RoboDK station: Silva_Honores_ProyectoFinal (1).rdk

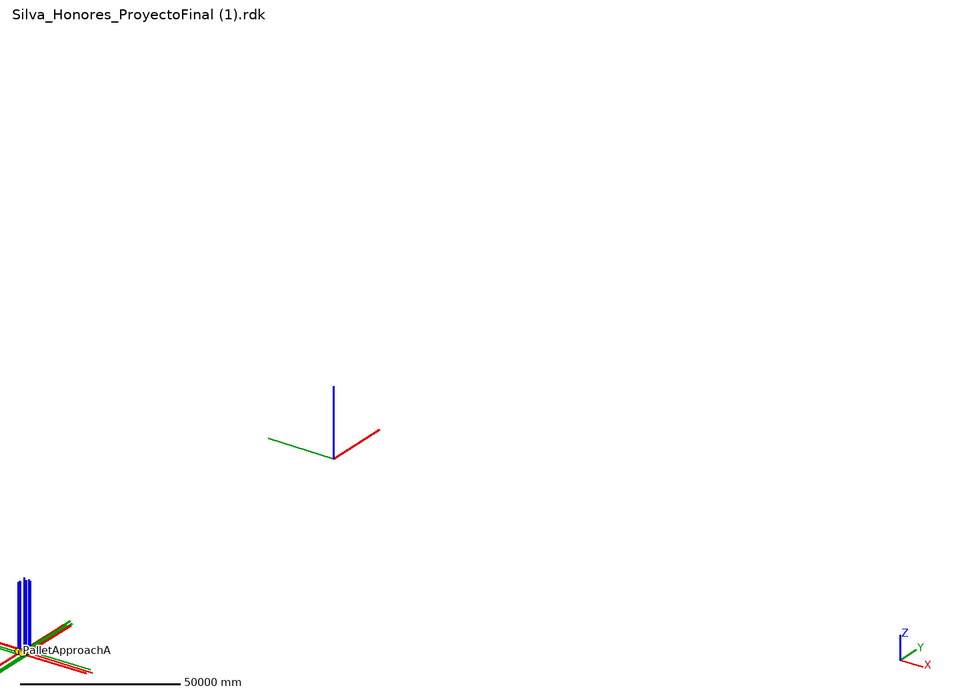
[picture v0: the station drawn from its stored meshes, robots at their saved joint values, targets as dots, program paths as lines]
Station Silva_Honores_ProyectoFinal (saved by RoboDK 5.3.0). Poses are relative to the parent item; angles as X-Y-Z fixed-axis rotations.
Station parameters (name, value as stored): SizeBox, 150, 200, 150, SizePallet, 3,2,3, ConvSpeed, 25.0, SENSOR, 0, verdes, 0, rojas, 0, azules, 0
  - frame Fanuc M-1iA/0.5SL Base at (787.66, 1086.23, 929.78) mm
    - robot Fanuc M-1iA/0.5SL: 4 axes, payload 0.5 kg, reach 420 mm, repeatability 0.03 mm, weight 23 kg
        joint limits [-25, -25, -25, -36000] to [80, 80, 80, 36000]; home [0, 0, 0, 0]; saved at [0, 0, 0, 0]
      - frame framecamera at (0, 0, 40) mm, rotated rx 0 ry 0 rz -90 deg
      - tool SICK VSPP-5f2113, TCP at (-100, 1870, 80) mm, rotated rx 0 ry 0 rz 90 deg, size 53 x 116 x 38 mm
  - frame UR10 Base A at (0, -212.57, -10) mm
    - robot UR10 A: 6 axes, payload 10 kg, reach 1300 mm, repeatability 0.1 mm, weight 28.9 kg
        modified DH rows (alpha deg, a mm, theta deg, d mm): 0, 0, 0, 118; 90, 0, 180, 0; 0, 612.7, 0, 0; 0, 571.6, 0, 163.9; -90, 0, 0, 115.7; 90, 0, 180, 92.2
        joint limits [-360, -360, -360, -360, -360, -360] to [360, 360, 360, 360, 360, 360]; home [0, -90, 90, -90, -90, 0]; saved at [152.649, -87.247, 87.177, -89.921, -90.005, -19.581]
      - tool GripperA, TCP at (0, 0, 30) mm, rotated rx 0 ry 0 rz 90 deg, size 209.9 x 42 x 100 mm, geometry from test.iges
    - frame PalletA at (-344.62, -460.78, -266.49) mm, rotated rx 0 ry 0 rz 90.24 deg
      - object Europallet at (0, 0, 0) mm, size 800 x 144 x 1200 mm, geometry from User Library-Europallet.igs
      - object box100mm at (0, 0, 0) mm, size 100 x 100 x 100 mm, geometry from box.sld
      - object Part 1 at (75, 100, 75) mm, size 150 x 200 x 150 mm, geometry from box.sld
      - object Part 2 at (225, 100, 75) mm, size 150 x 200 x 150 mm, geometry from box.sld
      - object Part 3 at (375, 100, 75) mm, size 150 x 200 x 150 mm, geometry from box.sld
      - object Part 4 at (75, 300, 75) mm, size 150 x 200 x 150 mm, geometry from box.sld
      - object Part 5 at (225, 300, 75) mm, size 150 x 200 x 150 mm, geometry from box.sld
      - object Part 6 at (375, 300, 75) mm, size 150 x 200 x 150 mm, geometry from box.sld
      - object Part 7 at (75, 100, 225) mm, size 150 x 200 x 150 mm, geometry from box.sld
      - object Part 8 at (225, 100, 225) mm, size 150 x 200 x 150 mm, geometry from box.sld
      - object Part 9 at (375, 100, 225) mm, size 150 x 200 x 150 mm, geometry from box.sld
      - object Part 10 at (75, 300, 225) mm, size 150 x 200 x 150 mm, geometry from box.sld
      - object Part 11 at (225, 300, 225) mm, size 150 x 200 x 150 mm, geometry from box.sld
      - object Part 12 at (375, 300, 225) mm, size 150 x 200 x 150 mm, geometry from box.sld
      - object Part 13 at (75, 100, 375) mm, size 150 x 200 x 150 mm, geometry from box.sld
      - object Part 14 at (225, 100, 375) mm, size 150 x 200 x 150 mm, geometry from box.sld
      - object Part 15 at (375, 100, 375) mm, size 150 x 200 x 150 mm, geometry from box.sld
      - object Part 16 at (75, 300, 375) mm, size 150 x 200 x 150 mm, geometry from box.sld
      - object Part 17 at (225, 300, 375) mm, size 150 x 200 x 150 mm, geometry from box.sld
      - object Part 18 at (375, 300, 375) mm, size 150 x 200 x 150 mm, geometry from box.sld
    - target PalletApproachA (joint target) at (-397.36, -413.15, 644.38) mm, rotated rx 180 ry 0 rz 88.83 deg; joints [29.502, -102.797, 97.668, -84.871, -90, -59.329] of UR10 A
    - target ConvApproachA (joint target) at (711.88, -183.71, 608.48) mm, rotated rx -180 ry -0.01 rz 172.23 deg; joints [152.649, -87.247, 87.177, -89.921, -90.005, -19.581] of UR10 A
  - frame UR10 Base B at (1478.64, 1242.75, 0) mm
    - robot UR10 B: 6 axes, payload 10 kg, reach 1300 mm, repeatability 0.1 mm, weight 28.9 kg
        modified DH rows (alpha deg, a mm, theta deg, d mm): 0, 0, 0, 118; 90, 0, 180, 0; 0, 612.7, 0, 0; 0, 571.6, 0, 163.9; -90, 0, 0, 115.7; 90, 0, 180, 92.2
        joint limits [-360, -360, -360, -360, -360, -360] to [360, 360, 360, 360, 360, 360]; home [0, -90, 90, -90, -90, 0]; saved at [262.56, -112.555, 122.685, -105, -90, 82.56]
      - tool GripperB, TCP at (0, 0, 30) mm, rotated rx 0 ry 0 rz 90 deg, size 209.9 x 42 x 100 mm, geometry from test.iges
    - target PalletApproachR (joint target) at (-103, 477.05, 396.64) mm, rotated rx 175.17 ry 0.63 rz 179.97 deg; joints [262.56, -112.555, 122.685, -105, -90, 82.56] of UR10 B
    - target ConvApproachB (joint target) at (-305.88, -163.9, 417.02) mm, rotated rx -180 ry 0 rz 0 deg; joints [0, -128.114, 134.225, -96.111, -90, 0] of UR10 B
    - target PalletApproachG (joint target) at (162.31, -616.99, 501.62) mm, rotated rx 176.81 ry 2.55 rz 88.83 deg; joints [88.829, -97.645, 100.863, -95.772, -86.806, 0] of UR10 B
    - target PalletApproachB (joint target) at (566.28, 157.58, 459.33) mm, rotated rx -180 ry 0 rz 179.36 deg; joints [-180.64, -99.905, 114.086, -104.182, -90, 0] of UR10 B
    - frame PalletB at (1076.11, 642.98, -166.38) mm, rotated rx 0 ry 0 rz 180 deg
      - object Europallet at (0, 0, 0) mm, size 800 x 144 x 1200 mm, geometry from User Library-Europallet.igs
    - frame PalletR at (254.08, 1192.65, -166.38) mm, rotated rx 0 ry 0 rz 180 deg
      - object Europallet at (0, 0, 13) mm, size 800 x 144 x 1200 mm, geometry from User Library-Europallet.igs
    - frame PalletG at (271.28, -1223.37, -166.38) mm, rotated rx 0 ry 0 rz 90 deg
      - object Europallet at (0, 800, 0) mm, rotated rx 0 ry 0 rz -90 deg, size 800 x 144 x 1200 mm, geometry from User Library-Europallet.igs
  - frame ConveyorReference at (597.23, -679.82, 119.18) mm
    - robot Conveyor Belt: 1 axes
        modified DH rows (alpha deg, a mm, theta deg, d mm): 0, 0, 0, 0 linear
        base shift (440, 200, 0) mm, rotated rx 0 ry 90 rz 90 deg
        joint limits [-500000] to [500000]; home [0]; saved at [169619]
      - frame MovingRef at (0, 0, 0) mm
    - target ConveyorHome (joint target) at (440, 200, 0) mm, rotated rx 0 ry 0 rz 90 deg; joints [0] of Conveyor Belt
    - target ConveyorMove (joint target) at (440, 500200, 0) mm, rotated rx 0 ry 0 rz 90 deg; joints [500000] of Conveyor Belt
    - object Sensor SICK WL4S at (504.09, 1950, 25) mm, rotated rx 90 ry 0 rz 180 deg, size 683.3 x 45.2 x 12.5 mm, geometry from SICK WL4S-3P1330-Order no.1042068 (1).stp
      - Python program SensorActivate (listed below)
    - target Get Conveyor (Cartesian target) at (200, 1900, 0) mm, rotated rx -180 ry 0 rz 0 deg; joints [-12.012, -70.873, 123.705, -142.833, -90, -12.012] of UR10 B
    - target Put Conveyor (Cartesian target) at (200, 422.12, 0) mm, rotated rx -180 ry 0 rz 180 deg; joints [164.915, -63.548, 110.129, -136.581, -90, -15.085] of UR10 A
  - Python program SetSimulationParams (listed below)
  - Python program PrepareSimulation (listed below)
  - Python program ProcesarColorBox (listed below)
  - Python program RobotA_GetParts (listed below)
  - Python program RobotB_StoreParts (listed below)
  - program MoveConveyor (1 instructions, listed below)
  - program MainSimulation (6 instructions, listed below)

--- Python program SensorActivate ---
#Ricardo Silva
#Steven Honores
#P101
from robolink import *    # API to communicate with RoboDK
from robodk import *      # basic matrix operations
RDK = Robolink()

# Use a target from the station as a reference plane:
SENSOR_NAME = 'Sensor SICK WL4S'
SENSOR_VARIABLE = 'SENSOR'

# Look for parts with the keyword "Part"
PART_KEYWORD = 'Part '

# Update status every 1 ms
RECHECK_PERIOD = 0.001

# Get the sensor and the detection plane
SENSOR = RDK.Item(SENSOR_NAME, ITEM_TYPE_OBJECT)

# retrieve all objects
all_objects = RDK.ItemList(ITEM_TYPE_OBJECT, False)
part_objects = []
for obj in all_objects:
    if obj.Name().count(PART_KEYWORD) > 0:
        part_objects.append(obj)


# Loop forever to detect parts
detected_status = -1
while True:
    detected = 0
    for obj in part_objects:
        # check if an object has the part keyword and is detected by the laser
        if SENSOR.Collision(obj) > 0:
            detected = 1
            break

    # update the current status of the sensor
    if detected_status != detected:
        detected_status = detected
        RDK.setParam(SENSOR_VARIABLE, detected_status)
        print('Object detected status --> %i' % detected_status)

    # Wait some time...
    pause(RECHECK_PERIOD)

--- Python program SetSimulationParams ---
#Ricardo Silva
#Steven Honores
#P101
from robolink import *    # API to communicate with RoboDK
from robodk import *      # basic matrix operations


PARAM_SIZE_BOX = 'SizeBox'
PARAM_SIZE_PALLET = 'SizePallet'
PARAM_CONV_SPEED_MM = 'ConvSpeed'



RDK = Robolink()

size_box = RDK.getParam(PARAM_SIZE_BOX)
size_pallet = RDK.getParam(PARAM_SIZE_PALLET)
conv_speed = RDK.getParam(PARAM_CONV_SPEED_MM)

# ------------------------------------------------------------
size_box_input = mbox('Enter the size of the box in mm [L,W,H]', entry=size_box)
if size_box_input:
    RDK.setParam(PARAM_SIZE_BOX, size_box_input)
else:
    raise Exception('Operation cancelled by user')

# ------------------------------------------------------------
size_pallet_input = mbox('Enter the size of the pallet', entry=size_pallet)
if size_pallet_input:
    RDK.setParam(PARAM_SIZE_PALLET, size_pallet_input)
else:
    raise Exception('Operation cancelled by user')

# ------------------------------------------------------------
conv_speed_input = mbox('Enter the speed of the conveyor in mm/s', entry=conv_speed)
if conv_speed_input:
    RDK.setParam(PARAM_CONV_SPEED_MM, conv_speed_input)
    conv_speed = float(conv_speed_input)
    conv = RDK.Item('Conveyor Belt', ITEM_TYPE_ROBOT)
    conv.setSpeed(conv_speed)

else:
    raise Exception('Operation cancelled by user')

--- Python program PrepareSimulation ---
#Ricardo Silva
#Steven Honores
#P101
from robolink import *    # API to communicate with RoboDK
from robodk import *      # basic matrix operations

import random   #importar libreria random
# Use RoboDK API as RL
RDK = Robolink()

frame_pallet        = RDK.Item('PalletA', ITEM_TYPE_FRAME)

# get variable parameters
SIZE_BOX = RDK.getParam('SizeBox')
SIZE_PALLET = RDK.getParam('SizePallet')
SIZE_BOX_XYZ = [float(x.replace(' ','')) for x in SIZE_BOX.split(',')]
SIZE_PALLET_XYZ = [float(x.replace(' ','')) for x in SIZE_PALLET.split(',')]
SIZE_BOX_Z = SIZE_BOX_XYZ[2] # the height of the boxes is important to take into account when approaching the positions

def box_calc(size_xyz, pallet_xyz):
    """Calculates a list of points to store parts in a pallet"""
    [size_x, size_y, size_z] = size_xyz
    [pallet_x, pallet_y, pallet_z] = pallet_xyz
    xyz_list = []
    for h in range(int(pallet_z)):
        for j in range(int(pallet_y)):
            for i in range(int(pallet_x)):
                xyz_list = xyz_list + [[(i+0.5)*size_x, (j+0.5)*size_y, (h+0.5)*size_z]]
    return xyz_list

def parts_setup(frame, positions, size_xyz):
    """Place a list of parts in a reference frame. The part/reference object must have been previously copied to the clipboard."""
    [size_x, size_y, size_z] = size_xyz
    nparts = len(positions)
    cstep = 1.0/(nparts - 1)
    color=0
    Mcolor=[]
    for i in range(nparts):
        newpart = frame.Paste()
        newpart.Scale([size_x/100, size_y/100, size_z/100]) #scale with respect to the reference object (100mm cube)
        newpart.setName('Part ' + str(i+1)) #set item name
        newpart.setPose(transl(positions[i])) #set item position with respect to parent
        newpart.setVisible(True, False) #make item visible but hide the reference frame
        #generacion de numeros aleatorios para cajas de colores aleatorios
        color = random.randint(0,2)
        Mcolor.append(color)
        if color==0:  #rojo
            newpart.setColor([1,0,0,1])
        elif color==1:  #verde
            newpart.setColor([0,1,0,1])
        elif color==2:  #azul
            newpart.setColor([0,0,1,1])
    print(Mcolor)

def cleanup(objects, startswith="Part "):
    """Deletes all objects where the name starts with "startswith", from the provided list of objects."""
    for item in objects:
        if item.Name().startswith(startswith):
            item.Delete()

# turn off rendering (much faster when setting up the station)
RDK.Render(False)

# cleanup previous simulation (generated parts and tools)
all_objects = RDK.ItemList(ITEM_TYPE_OBJECT, False)
cleanup(all_objects, 'Part ')
all_tools = RDK.ItemList(ITEM_TYPE_TOOL, False)
cleanup(all_tools, 'TCP ')

# copy the reference part
partref = RDK.Item('box100mm')
partref.Copy()

# calculate an array of positions to get/store the parts
parts_positions = box_calc(SIZE_BOX_XYZ, SIZE_PALLET_XYZ)

# setup/initialise the parts on the palled
parts_setup(frame_pallet, parts_positions, SIZE_BOX_XYZ)

RDK.Render(True)

--- Python program ProcesarColorBox ---
#Ricardo Silva
#Steven Honores
#P101
from time import sleep
from robodk import *
from robolink import *
import datetime

from tkinter import *
from tkinter import filedialog

####procesamiento de imagen###
import cv2
import numpy as np
RDK = Robolink()


while(1):

    VERDES = 'verdes'
    RDK.setParam(VERDES,0)
    ROJAS = 'rojas'
    RDK.setParam(ROJAS,0)
    AZULES = 'azules'
    RDK.setParam(AZULES,0)

    SENSOR_VARIABLE = 'SENSOR'

    path_rdk = RDK.getParam('PATH_OPENSTATION')
    file_name = "/foto.jpg" #"RoboDK-Screenshot-HQ-" + date_str + ".png"

    root = Tk()
    root.withdraw()

    #RDK.Render(False) # prevent flickering

    # select a reference frame at the camera view location
    ref_cam = RDK.Item("framecamera",ITEM_TYPE_FRAME)
    ref_cam.setVisible(False)

    cam_id = RDK.Cam2D_Add(ref_cam, 'FOCAL_LENGHT=6 FOV=32 FAR_LENGHT=200 SIZE=320x240 BG_COLOR=black')

    ####procesamiento de imagen###
    def WaitSensor():
        if RDK.RunMode() == RUNMODE_SIMULATE:
            # Simulate the sensor by waiting for the SENSOR status to turn to 1 (object present)
            while RDK.getParam(SENSOR_VARIABLE) == 0:
                pause(0.001)
        else:
            RDK.RunProgram('WaitSensor')
        print("Part detected")

    WaitSensor()

    RDK.Cam2D_Snapshot((path_rdk+file_name), cam_id)
    print(path_rdk+file_name)
    RDK.Cam2D_Close(cam_id)

    # Delete the temporary reference added
    #ref_cam.Delete()
    cam_id.Delete()
    print("Done")
    #RDK.ShowMessage("High resolution snapshot saved: " + file_path, False)

    img = cv2.imdecode(np.fromfile(path_rdk+file_name, dtype=np.uint8), cv2.IMREAD_UNCHANGED)
    print(img.shape)

    imagenHSV = cv2.cvtColor(img, cv2.COLOR_BGR2HSV)

    ##verdes
    verdeBajo = np.array([36, 100, 20], np.uint8)
    verdeAlto = np.array([70, 255, 255], np.uint8)
    maskVerde = cv2.inRange(imagenHSV, verdeBajo, verdeAlto)
    ##verdes

    ##rojos
    rojoBajo1 = np.array([0, 100, 20], np.uint8)
    rojoAlto1 = np.array([10, 255, 255], np.uint8)
    rojoBajo2 = np.array([175, 100, 20], np.uint8)
    rojoAlto2 = np.array([180, 255, 255], np.uint8)

    maskRojo1 = cv2.inRange(imagenHSV, rojoBajo1, rojoAlto1)
    maskRojo2 = cv2.inRange(imagenHSV, rojoBajo2, rojoAlto2)
    maskRojo =  cv2.add(maskRojo1, maskRojo2)
    ##rojos

    ##azul
    azul_bajos = np.array([40,0,0])
    azul_altos = np.array([255,120,120])
    maskazul = cv2.inRange(img, azul_bajos, azul_altos)
    ##azul

    contornosazul,oooooo1 = cv2.findContours(maskazul, cv2.RETR_TREE, cv2.CHAIN_APPROX_SIMPLE)
    print("contornos azules",len(contornosazul))

    contornosrojo,oooooo2 = cv2.findContours(maskRojo, cv2.RETR_TREE, cv2.CHAIN_APPROX_SIMPLE)
    print("contornos rojo",len(contornosrojo))

    contornosverde,oooooo3 = cv2.findContours(maskVerde, cv2.RETR_TREE, cv2.CHAIN_APPROX_SIMPLE)
    print("contornos verde",len(contornosverde))

    ##enumerando por color
    #RDK.ShowMessage("%s " %len(contornosazul)+"azules, " +"%s " %len(contornosrojo)+"rojos, " +"%s " %len(contornosverde)+"verdes",False)

    RDK.setParam(VERDES,len(contornosverde))

    RDK.setParam(ROJAS,len(contornosrojo))

    RDK.setParam(AZULES,len(contornosazul))

    def WaitSensorDes():
        if RDK.RunMode() == RUNMODE_SIMULATE:
            # Simulate the sensor by waiting for the SENSOR status to turn to 1 (object present)
            while RDK.getParam(SENSOR_VARIABLE) == 1:
                pause(0.001)
        else:
            RDK.RunProgram('WaitSensorDes')
        print("Part detected")

    WaitSensorDes()

--- Python program RobotA_GetParts ---
#Ricardo Silva
#Steven Honores
#P101
from robolink import *    # API to communicate with RoboDK
from robodk import *      # basic matrix operations

# Use RoboDK API as RL
RDK = Robolink()

# define default approach distance
APPROACH = 100

# gather robot, tool and reference frames from the station
robot               = RDK.Item('UR10 A', ITEM_TYPE_ROBOT)
tool                = RDK.Item('GripperA', ITEM_TYPE_TOOL)
frame_pallet        = RDK.Item('PalletA', ITEM_TYPE_FRAME)
frame_conv          = RDK.Item('ConveyorReference', ITEM_TYPE_FRAME)
frame_conv_moving   = RDK.Item('MovingRef', ITEM_TYPE_FRAME)

# gather targets
target_pallet_safe = RDK.Item('PalletApproachA', ITEM_TYPE_TARGET)
target_conv_safe = RDK.Item('ConvApproachA', ITEM_TYPE_TARGET)
target_conv = RDK.Item('Put Conveyor', ITEM_TYPE_TARGET)

# get variable parameters
SIZE_BOX = RDK.getParam('SizeBox')
SIZE_PALLET = RDK.getParam('SizePallet')
SIZE_BOX_XYZ = [float(x.replace(' ','')) for x in SIZE_BOX.split(',')]
SIZE_PALLET_XYZ = [float(x.replace(' ','')) for x in SIZE_PALLET.split(',')]
SIZE_BOX_Z = SIZE_BOX_XYZ[2] # the height of the boxes is important to take into account when approaching the positions

def box_calc(size_xyz, pallet_xyz):
    """Calculates a list of points to store parts in a pallet"""
    [size_x, size_y, size_z] = size_xyz
    [pallet_x, pallet_y, pallet_z] = pallet_xyz
    xyz_list = []
    for h in range(int(pallet_z)):
        for j in range(int(pallet_y)):
            for i in range(int(pallet_x)):
                xyz_list = xyz_list + [[(i+0.5)*size_x, (j+0.5)*size_y, (h+0.5)*size_z]]
    return xyz_list

def TCP_On(toolitem):
    """Attaches the closest object to the toolitem Htool pose,
    It will also output appropriate function calls on the generated robot program (call to TCP_On)"""
    toolitem.AttachClosest()
    toolitem.RDK().RunMessage('Set air valve on')
    toolitem.RDK().RunProgram('TCP_On()');

def TCP_Off(toolitem, itemleave=0):
    """Detaches the closest object attached to the toolitem Htool pose,
    It will also output appropriate function calls on the generated robot program (call to TCP_Off)"""
    toolitem.DetachAll(itemleave)
    toolitem.RDK().RunMessage('Set air valve off')
    toolitem.RDK().RunProgram('TCP_Off()');

#RL.Set_Simulation_Speed(500);
#RL.Set_Simulation_Mode(1)

# calculate an array of positions to get/store the parts
parts_positions = box_calc(SIZE_BOX_XYZ, SIZE_PALLET_XYZ)

# Calculate a new TCP that takes into account the size of the part (targets are set to the center of the box)
tool_xyzrpw = tool.PoseTool()*transl(0,0,SIZE_BOX_Z/2)
tool_tcp = robot.AddTool(tool_xyzrpw, 'TCP A')

# ---------------------------------------------------------------------------------
# -------------------------- PROGRAM START ----------------------------------------

robot.setPoseTool(tool_tcp)
nparts = len(parts_positions)
i = nparts-1
while i >= 0:
    # ----------- take a part from the pallet ------
    # get the xyz position of part i
    robot.setPoseFrame(frame_pallet)
    part_position_i = parts_positions[i]
    target_i = transl(part_position_i)*rotx(pi)
    target_i_app = target_i * transl(0,0,-(APPROACH+SIZE_BOX_Z))
    # approach to the pallet
    robot.MoveJ(target_pallet_safe)
    # get the box i
    robot.MoveJ(target_i_app)
    robot.MoveL(target_i)
    TCP_On(tool) # attach the closest part
    robot.MoveL(target_i_app)
    robot.MoveJ(target_pallet_safe)

    # ----------- place the box i on the convegor ------
    # approach to the conveyor
    robot.setPoseFrame(frame_conv)
    target_conv_pose = target_conv.Pose()*transl(0,0,-SIZE_BOX_Z/2)
    target_conv_app = target_conv_pose*transl(0,0,-APPROACH)
    robot.MoveJ(target_conv_safe)
    robot.MoveJ(target_conv_app)
    robot.MoveL(target_conv_pose)
    TCP_Off(tool, frame_conv_moving) # detach an place the object in the moving reference frame of the conveyor
    robot.MoveL(target_conv_app)
    robot.MoveJ(target_conv_safe)

    i = i - 1

--- Python program RobotB_StoreParts ---
#Ricardo Silva
#Steven Honores
#P101
from robolink import *    # API to communicate with RoboDK
from robodk import *      # basic matrix operations

# Use RoboDK API as RL
RDK = Robolink()

# define default approach distance
APPROACH = 100
SENSOR_VARIABLE = 'SENSOR' # station variable
VERDES = 'verdes'    #Variable de estacion
ROJAS = 'rojas'      #Variable de estacion
AZULES = 'azules'    #Variable de estacion

# gather robot, tool and reference frames from the station
robot               = RDK.Item('UR10 B', ITEM_TYPE_ROBOT)
tool                = RDK.Item('GripperB', ITEM_TYPE_TOOL)
#frame_pallet        = RDK.Item('PalletB', ITEM_TYPE_FRAME)      #Aqui se manda la caja al pallet B  !!!!!! Originalmente estaba en PalletB
frame_conv          = RDK.Item('ConveyorReference', ITEM_TYPE_FRAME)
frame_conv_moving   = RDK.Item('MovingRef', ITEM_TYPE_FRAME)

# gather targets
#target_pallet_safe = RDK.Item('PalletApproachB', ITEM_TYPE_TARGET)      #Aqui se manda el target del pallet a dejar la caja !!!!!!!  Originalmente estaba en PalletApproachB
target_conv_safe = RDK.Item('ConvApproachB', ITEM_TYPE_TARGET)
target_conv = RDK.Item('Get Conveyor', ITEM_TYPE_TARGET)

# get variable parameters
SIZE_BOX = RDK.getParam('SizeBox')
SIZE_PALLET = RDK.getParam('SizePallet')
SIZE_BOX_XYZ = [float(x.replace(' ','')) for x in SIZE_BOX.split(',')]
SIZE_PALLET_XYZ = [float(x.replace(' ','')) for x in SIZE_PALLET.split(',')]
SIZE_BOX_Z = SIZE_BOX_XYZ[2] # the height of the boxes is important to take into account when approaching the positions

def box_calc(size_xyz, pallet_xyz):
    """Calculates a list of points to store parts in a pallet"""
    [size_x, size_y, size_z] = size_xyz
    [pallet_x, pallet_y, pallet_z] = pallet_xyz
    xyz_list = []
    for h in range(int(pallet_z)):
        for j in range(int(pallet_y)):
            for i in range(int(pallet_x)):
                xyz_list = xyz_list + [[(i+0.5)*size_x, (j+0.5)*size_y, (h+0.5)*size_z]]
    return xyz_list

def TCP_On(toolitem):
    """Attaches the closest object to the toolitem Htool pose,
    It will also output appropriate function calls on the generated robot program (call to TCP_On)"""
    toolitem.AttachClosest()
    toolitem.RDK().RunMessage('Set air valve on')
    toolitem.RDK().RunProgram('TCP_On()');

def TCP_Off(toolitem, itemleave=0):
    """Detaches the closest object attached to the toolitem Htool pose,
    It will also output appropriate function calls on the generated robot program (call to TCP_Off)"""
    #toolitem.DetachClosest(itemleave)
    toolitem.DetachAll(itemleave)
    toolitem.RDK().RunMessage('Set air valve off')
    toolitem.RDK().RunProgram('TCP_Off()');

# calculate an array of positions to get/store the parts
parts_positions = box_calc(SIZE_BOX_XYZ, SIZE_PALLET_XYZ)

# Calculate a new TCP that takes into account the size of the part (targets are set to the center of the box)
tool_xyzrpw = tool.PoseTool()*transl(0,0,SIZE_BOX_Z/2)
tool_tcp = robot.AddTool(tool_xyzrpw, 'TCP B')

# ---------------------------------------------------------------------------------
# -------------------------- PROGRAM START ----------------------------------------

def WaitSensor():
    if RDK.RunMode() == RUNMODE_SIMULATE:
        # Simulate the sensor by waiting for the SENSOR status to turn to 1 (object present)
        while RDK.getParam(SENSOR_VARIABLE) == 0:
            pause(0.001)
    else:
        RDK.RunProgram('WaitSensor')
    print("Part detected")
    print('R',RDK.getParam(ROJAS))  #!!!
    print('A',RDK.getParam(AZULES))    #!!!!
    print('V',RDK.getParam(VERDES))    #!!!!!
    #-------------determinar a que pallet el robot llevara la caja por su color------------      #aqui se hace la validacion de que color es  RDK.getParam(VERDES)==1

def DecidirPallet():     #Funcion creada para organizar las cajas por colores
    frame_pallet = RDK.Item('PalletR', ITEM_TYPE_FRAME)  #por default
    target_pallet_safe = RDK.Item('PalletApproachR', ITEM_TYPE_TARGET)   #por default
    if RDK.getParam(ROJAS) == 1.0:  #rojo
        frame_pallet = RDK.Item('PalletR', ITEM_TYPE_FRAME)
        target_pallet_safe = RDK.Item('PalletApproachR', ITEM_TYPE_TARGET)

    elif RDK.getParam(VERDES) == 1.0:  #verde
        frame_pallet = RDK.Item('PalletG', ITEM_TYPE_FRAME)
        target_pallet_safe = RDK.Item('PalletApproachG', ITEM_TYPE_TARGET)

    elif RDK.getParam(AZULES) == 1.0:  #azul
        frame_pallet = RDK.Item('PalletB', ITEM_TYPE_FRAME)
        target_pallet_safe = RDK.Item('PalletApproachB', ITEM_TYPE_TARGET)

    return frame_pallet,target_pallet_safe

robot.setPoseTool(tool_tcp)
nparts = len(parts_positions)
i = 0
irojo = 0
iazul = 0
iverde = 0
x = 0

while i < nparts:

    # ----------- place the box i on the convegor ------
    # approach to the conveyor
    robot.setPoseFrame(frame_conv)
    target_conv_pose = target_conv.Pose()*transl(0,0,-SIZE_BOX_Z/2)
    target_conv_app = target_conv_pose*transl(0,0,-APPROACH)
    robot.MoveJ(target_conv_safe)
    robot.MoveJ(target_conv_app)
    WaitSensor()
    frame_pallet,target_pallet_safe=DecidirPallet()   #Aqui se valida la funcion que determina el pallet a colocar la caja por su color
    robot.MoveL(target_conv_pose)
    TCP_On(tool) # detach an place the object in the moving reference frame of the conveyor
    robot.MoveL(target_conv_app)
    robot.MoveJ(target_conv_safe)

    if frame_pallet == RDK.Item('PalletB', ITEM_TYPE_FRAME):
        x = iazul
        iazul= iazul + 1
    elif frame_pallet == RDK.Item('PalletG', ITEM_TYPE_FRAME):
        x = iverde
        iverde= iverde + 1
    elif frame_pallet == RDK.Item('PalletR', ITEM_TYPE_FRAME):
        x = irojo
        irojo= irojo + 1



    # ----------- take a part from the conveyor ------
    # get the xyz position of part i
    robot.setPoseFrame(frame_pallet)
    part_position_i = parts_positions[x]
    target_i = transl(part_position_i)*rotx(pi)
    target_i_app = target_i * transl(0,0,-(APPROACH+SIZE_BOX_Z))
    # approach to the pallet
    robot.MoveJ(target_pallet_safe)
    # get the box i
    robot.MoveJ(target_i_app)
    robot.MoveL(target_i)
    TCP_Off(tool, frame_pallet) # attach the closest part
    robot.MoveL(target_i_app)
    robot.MoveJ(target_pallet_safe)

    i = i + 1

--- program MoveConveyor (robot Conveyor Belt) ---
  MoveJ (ConveyorMove)

--- program MainSimulation (robot UR10 A) ---
  Call PrepareSimulation
  Run MoveConveyor
  Run RobotA_GetParts
  Run SensorActivate
  Run ProcesarColorBox
  Call RobotB_StoreParts
